// TIA Portal V17 export
// export: Created 2024-08-29T18:23:44.0966443Z, ExportSetting WithDefaults, DisplayName Totally Integrated Automation Portal, DisplayVersion V17 Update 7, DisplayName TIA Portal Openness, DisplayVersion V17 Update 7, DisplayName TIA Portal Version Control Interface, DisplayVersion V17, DisplayName SINAMICS Startdrive Advanced, DisplayVersion V17 SP2, DisplayName SINAMICS Startdrive G110M, G120, G120C, G120D, G120P, G115D, DisplayVersion V17 SP2, DisplayName SINAMICS Startdrive G130, G150, S120, S150, SINAMICS MV, S210, DisplayVersion V17 SP2, DisplayName STEP 7 Professional, DisplayVersion V17 Update 7, DisplayName STEP 7 Safety, DisplayVersion V17 Update 6, DisplayName WinCC Advanced / Unified PC, DisplayVersion V17 Update 7
FUNCTION "cylinderControl" : Void   // FC9, LAD
{ S7_Optimized_Access := 'TRUE' }
VERSION : 0.1
// stored: AutoNumber true, IsIECCheckEnabled false, SetENOAutomatically false, UDAEnableTagReadback false
   VAR_TEMP
      leftTrackReady : Bool;
      rightTrackReady : Bool;
      plasticBridgeReady : Bool;
      retractLocatingPinReady : Bool;
      enableCylinders : Bool;
      retractClampsReady : Bool;
   END_VAR
   VAR_TEMP   // added for the SCL form of the ladder/FBD networks
      _w1 : Bool;
   END_VAR
BEGIN

REGION Network 1: ENABLE CYLINDER GLOBAL
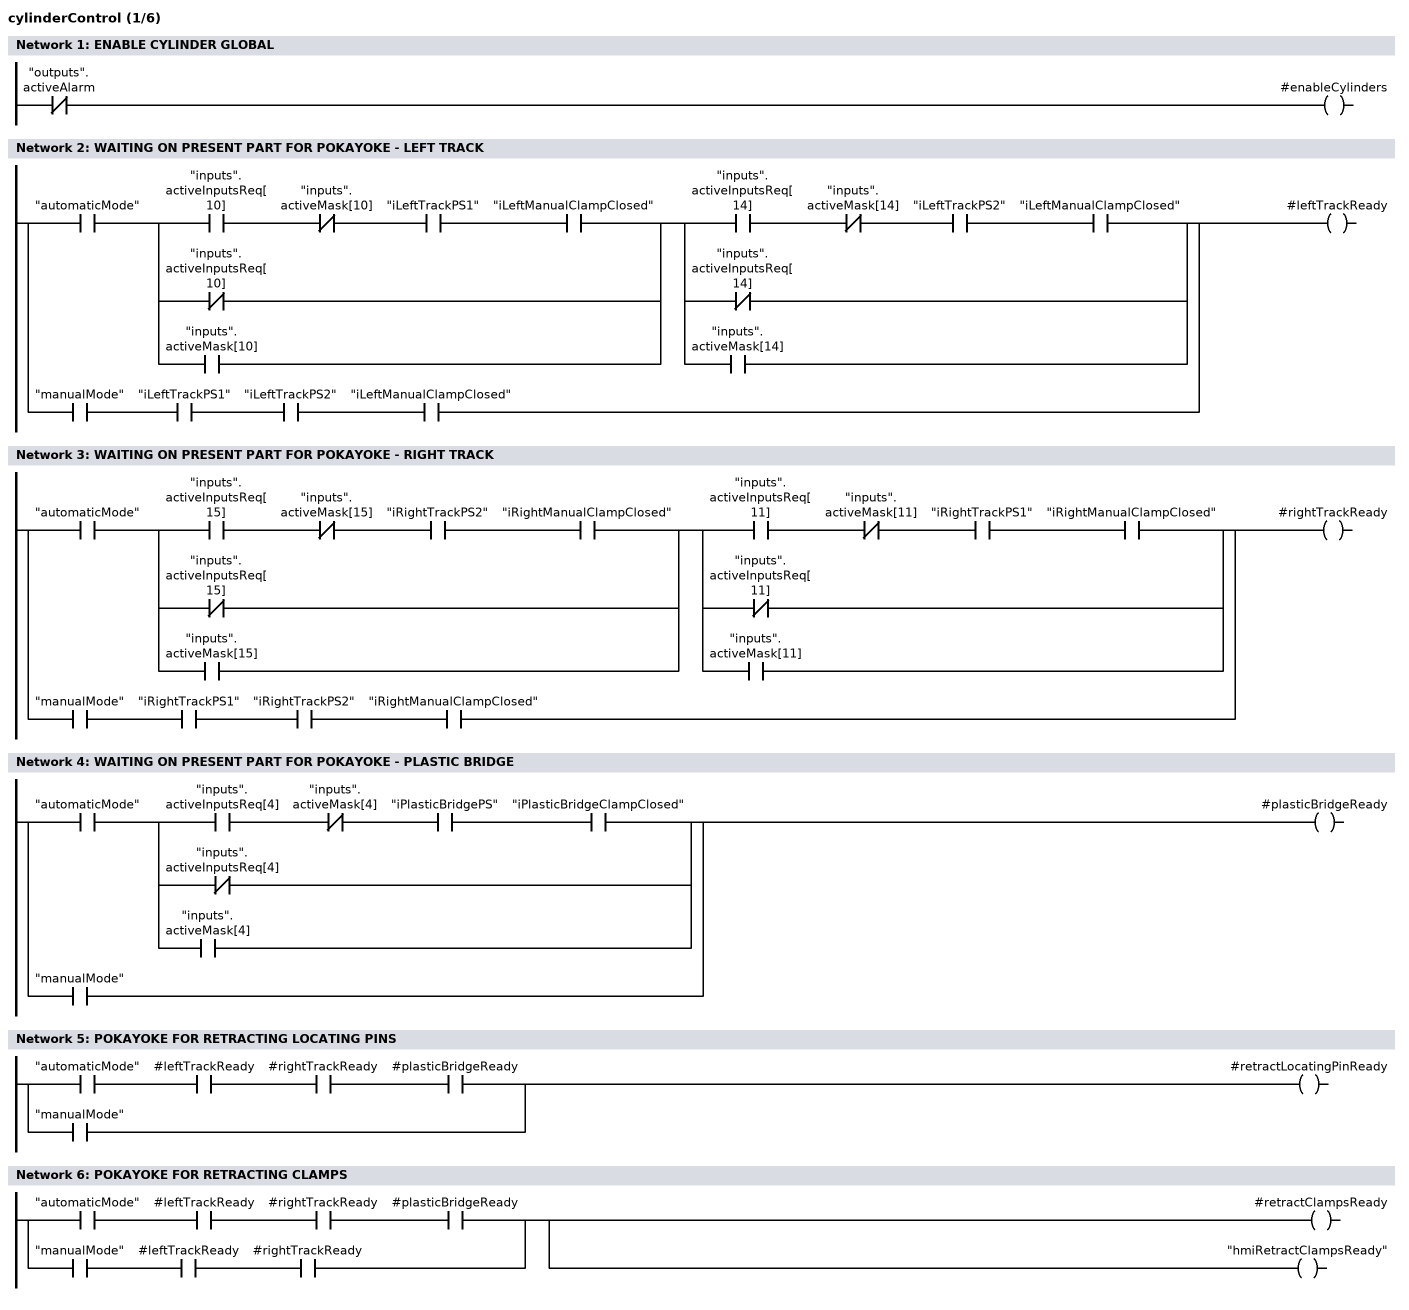
   RUNG wire#powerrail
      I_Contact( "outputs".activeAlarm )
      Coil( #enableCylinders )
   END_RUNG
   // the same network as SCL:
   #enableCylinders := NOT "outputs".activeAlarm;
END_REGION

REGION Network 2: WAITING ON PRESENT PART FOR POKAYOKE - LEFT TRACK
   RUNG wire#powerrail
      Contact( "automaticMode" )
      wire#w1
      Contact( "inputs".activeInputsReq[10] )
      I_Contact( "inputs".activeMask[10] )
      Contact( "iLeftTrackPS1" )
      Contact( "iLeftManualClampClosed" )
      wire#w2
      Contact( "inputs".activeInputsReq[14] )
      I_Contact( "inputs".activeMask[14] )
      Contact( "iLeftTrackPS2" )
      Contact( "iLeftManualClampClosed" )
      wire#w3
      Coil( #leftTrackReady )
   END_RUNG
   RUNG wire#w1
      I_Contact( "inputs".activeInputsReq[10] )
   END_RUNG wire#w2
   RUNG wire#w1
      Contact( "inputs".activeMask[10] )
   END_RUNG wire#w2
   RUNG wire#w2
      I_Contact( "inputs".activeInputsReq[14] )
   END_RUNG wire#w3
   RUNG wire#w2
      Contact( "inputs".activeMask[14] )
   END_RUNG wire#w3
   RUNG wire#powerrail
      Contact( "manualMode" )
      Contact( "iLeftTrackPS1" )
      Contact( "iLeftTrackPS2" )
      Contact( "iLeftManualClampClosed" )
   END_RUNG wire#w3
   // the same network as SCL:
   #leftTrackReady := ("automaticMode" AND (("inputs".activeInputsReq[10] AND NOT "inputs".activeMask[10] AND "iLeftTrackPS1" AND "iLeftManualClampClosed") OR NOT "inputs".activeInputsReq[10] OR "inputs".activeMask[10]) AND (("inputs".activeInputsReq[14] AND NOT "inputs".activeMask[14] AND "iLeftTrackPS2" AND "iLeftManualClampClosed") OR NOT "inputs".activeInputsReq[14] OR "inputs".activeMask[14])) OR ("manualMode" AND "iLeftTrackPS1" AND "iLeftTrackPS2" AND "iLeftManualClampClosed");
END_REGION

REGION Network 3: WAITING ON PRESENT PART FOR POKAYOKE - RIGHT TRACK
   RUNG wire#powerrail
      Contact( "automaticMode" )
      wire#w1
      Contact( "inputs".activeInputsReq[15] )
      I_Contact( "inputs".activeMask[15] )
      Contact( "iRightTrackPS2" )
      Contact( "iRightManualClampClosed" )
      wire#w2
      Contact( "inputs".activeInputsReq[11] )
      I_Contact( "inputs".activeMask[11] )
      Contact( "iRightTrackPS1" )
      Contact( "iRightManualClampClosed" )
      wire#w3
      Coil( #rightTrackReady )
   END_RUNG
   RUNG wire#w1
      I_Contact( "inputs".activeInputsReq[15] )
   END_RUNG wire#w2
   RUNG wire#w1
      Contact( "inputs".activeMask[15] )
   END_RUNG wire#w2
   RUNG wire#w2
      I_Contact( "inputs".activeInputsReq[11] )
   END_RUNG wire#w3
   RUNG wire#w2
      Contact( "inputs".activeMask[11] )
   END_RUNG wire#w3
   RUNG wire#powerrail
      Contact( "manualMode" )
      Contact( "iRightTrackPS1" )
      Contact( "iRightTrackPS2" )
      Contact( "iRightManualClampClosed" )
   END_RUNG wire#w3
   // the same network as SCL:
   #rightTrackReady := ("automaticMode" AND (("inputs".activeInputsReq[15] AND NOT "inputs".activeMask[15] AND "iRightTrackPS2" AND "iRightManualClampClosed") OR NOT "inputs".activeInputsReq[15] OR "inputs".activeMask[15]) AND (("inputs".activeInputsReq[11] AND NOT "inputs".activeMask[11] AND "iRightTrackPS1" AND "iRightManualClampClosed") OR NOT "inputs".activeInputsReq[11] OR "inputs".activeMask[11])) OR ("manualMode" AND "iRightTrackPS1" AND "iRightTrackPS2" AND "iRightManualClampClosed");
END_REGION

REGION Network 4: WAITING ON PRESENT PART FOR POKAYOKE - PLASTIC BRIDGE
   RUNG wire#powerrail
      Contact( "automaticMode" )
      wire#w1
      Contact( "inputs".activeInputsReq[4] )
      I_Contact( "inputs".activeMask[4] )
      Contact( "iPlasticBridgePS" )
      Contact( "iPlasticBridgeClampClosed" )
      wire#w2
      Coil( #plasticBridgeReady )
   END_RUNG
   RUNG wire#w1
      I_Contact( "inputs".activeInputsReq[4] )
   END_RUNG wire#w2
   RUNG wire#w1
      Contact( "inputs".activeMask[4] )
   END_RUNG wire#w2
   RUNG wire#powerrail
      Contact( "manualMode" )
   END_RUNG wire#w2
   // the same network as SCL:
   #plasticBridgeReady := ("automaticMode" AND (("inputs".activeInputsReq[4] AND NOT "inputs".activeMask[4] AND "iPlasticBridgePS" AND "iPlasticBridgeClampClosed") OR NOT "inputs".activeInputsReq[4] OR "inputs".activeMask[4])) OR "manualMode";
END_REGION

REGION Network 5: POKAYOKE FOR RETRACTING LOCATING PINS
   RUNG wire#powerrail
      Contact( "automaticMode" )
      Contact( #leftTrackReady )
      Contact( #rightTrackReady )
      Contact( #plasticBridgeReady )
      wire#w1
      Coil( #retractLocatingPinReady )
   END_RUNG
   RUNG wire#powerrail
      Contact( "manualMode" )
   END_RUNG wire#w1
   // the same network as SCL:
   #retractLocatingPinReady := ("automaticMode" AND #leftTrackReady AND #rightTrackReady AND #plasticBridgeReady) OR "manualMode";
END_REGION

REGION Network 6: POKAYOKE FOR RETRACTING CLAMPS
   RUNG wire#powerrail
      Contact( "automaticMode" )
      Contact( #leftTrackReady )
      Contact( #rightTrackReady )
      Contact( #plasticBridgeReady )
      wire#w1
      Coil( #retractClampsReady )
   END_RUNG
   RUNG wire#powerrail
      Contact( "manualMode" )
      Contact( #leftTrackReady )
      Contact( #rightTrackReady )
   END_RUNG wire#w1
   RUNG wire#w1
      Coil( "hmiRetractClampsReady" )
   END_RUNG
   // the same network as SCL:
   #retractClampsReady := ("automaticMode" AND #leftTrackReady AND #rightTrackReady AND #plasticBridgeReady) OR ("manualMode" AND #leftTrackReady AND #rightTrackReady);
   "hmiRetractClampsReady" := #retractClampsReady;
END_REGION

REGION Network 7: EXT CYL 1.- LEFT NEST LOCATING PIN EXTENDED
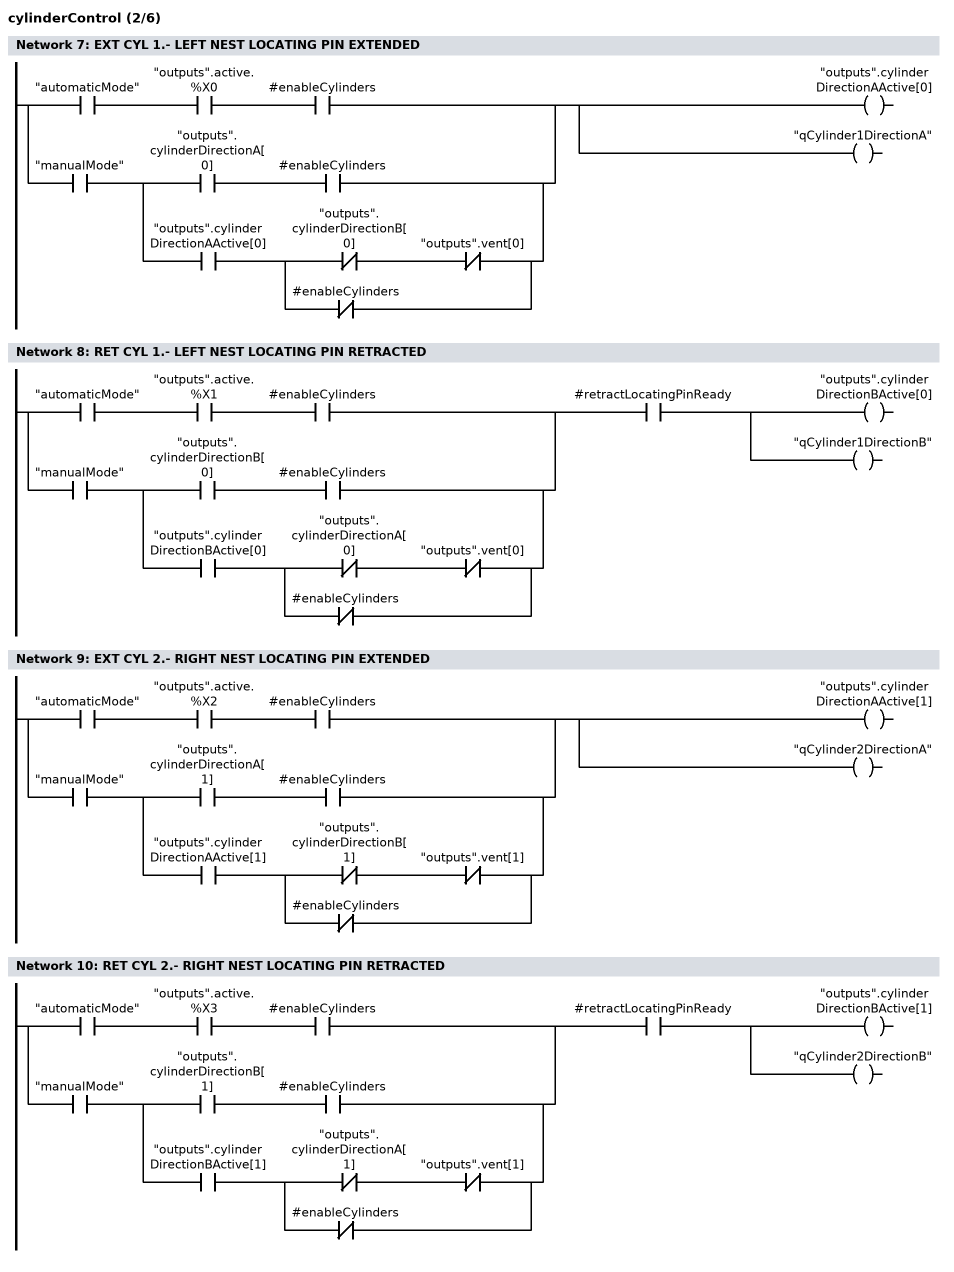
   RUNG wire#powerrail
      Contact( "automaticMode" )
      Contact( "outputs".active.%X0 )
      Contact( #enableCylinders )
      wire#w1
      Coil( "outputs".cylinderDirectionAActive[0] )
   END_RUNG
   RUNG wire#powerrail
      Contact( "manualMode" )
      wire#w2
      Contact( "outputs".cylinderDirectionA[0] )
      Contact( #enableCylinders )
   END_RUNG wire#w1
   RUNG wire#w2
      Contact( "outputs".cylinderDirectionAActive[0] )
      wire#w3
      I_Contact( "outputs".cylinderDirectionB[0] )
      I_Contact( "outputs".vent[0] )
   END_RUNG wire#w1
   RUNG wire#w3
      I_Contact( #enableCylinders )
   END_RUNG wire#w1
   RUNG wire#w1
      Coil( "qCylinder1DirectionA" )
   END_RUNG
   // the same network as SCL:
   #_w1 := ("automaticMode" AND "outputs".active.%X0 AND #enableCylinders) OR ("manualMode" AND (("outputs".cylinderDirectionA[0] AND #enableCylinders) OR ("outputs".cylinderDirectionAActive[0] AND ((NOT "outputs".cylinderDirectionB[0] AND NOT "outputs".vent[0]) OR NOT #enableCylinders))));
   "outputs".cylinderDirectionAActive[0] := ("automaticMode" AND "outputs".active.%X0 AND #enableCylinders) OR ("manualMode" AND (("outputs".cylinderDirectionA[0] AND #enableCylinders) OR ("outputs".cylinderDirectionAActive[0] AND ((NOT "outputs".cylinderDirectionB[0] AND NOT "outputs".vent[0]) OR NOT #enableCylinders))));
   "qCylinder1DirectionA" := #_w1;
END_REGION

REGION Network 8: RET CYL 1.- LEFT NEST LOCATING PIN RETRACTED
   RUNG wire#powerrail
      Contact( "automaticMode" )
      Contact( "outputs".active.%X1 )
      Contact( #enableCylinders )
      wire#w1
      Contact( #retractLocatingPinReady )
      wire#w4
      Coil( "outputs".cylinderDirectionBActive[0] )
   END_RUNG
   RUNG wire#powerrail
      Contact( "manualMode" )
      wire#w2
      Contact( "outputs".cylinderDirectionB[0] )
      Contact( #enableCylinders )
   END_RUNG wire#w1
   RUNG wire#w2
      Contact( "outputs".cylinderDirectionBActive[0] )
      wire#w3
      I_Contact( "outputs".cylinderDirectionA[0] )
      I_Contact( "outputs".vent[0] )
   END_RUNG wire#w1
   RUNG wire#w3
      I_Contact( #enableCylinders )
   END_RUNG wire#w1
   RUNG wire#w4
      Coil( "qCylinder1DirectionB" )
   END_RUNG
   // the same network as SCL:
   #_w1 := (("automaticMode" AND "outputs".active.%X1 AND #enableCylinders) OR ("manualMode" AND (("outputs".cylinderDirectionB[0] AND #enableCylinders) OR ("outputs".cylinderDirectionBActive[0] AND ((NOT "outputs".cylinderDirectionA[0] AND NOT "outputs".vent[0]) OR NOT #enableCylinders))))) AND #retractLocatingPinReady;
   "outputs".cylinderDirectionBActive[0] := (("automaticMode" AND "outputs".active.%X1 AND #enableCylinders) OR ("manualMode" AND (("outputs".cylinderDirectionB[0] AND #enableCylinders) OR ("outputs".cylinderDirectionBActive[0] AND ((NOT "outputs".cylinderDirectionA[0] AND NOT "outputs".vent[0]) OR NOT #enableCylinders))))) AND #retractLocatingPinReady;
   "qCylinder1DirectionB" := #_w1;
END_REGION

REGION Network 9: EXT CYL 2.- RIGHT NEST LOCATING PIN EXTENDED
   RUNG wire#powerrail
      Contact( "automaticMode" )
      Contact( "outputs".active.%X2 )
      Contact( #enableCylinders )
      wire#w1
      Coil( "outputs".cylinderDirectionAActive[1] )
   END_RUNG
   RUNG wire#powerrail
      Contact( "manualMode" )
      wire#w2
      Contact( "outputs".cylinderDirectionA[1] )
      Contact( #enableCylinders )
   END_RUNG wire#w1
   RUNG wire#w2
      Contact( "outputs".cylinderDirectionAActive[1] )
      wire#w3
      I_Contact( "outputs".cylinderDirectionB[1] )
      I_Contact( "outputs".vent[1] )
   END_RUNG wire#w1
   RUNG wire#w3
      I_Contact( #enableCylinders )
   END_RUNG wire#w1
   RUNG wire#w1
      Coil( "qCylinder2DirectionA" )
   END_RUNG
   // the same network as SCL:
   #_w1 := ("automaticMode" AND "outputs".active.%X2 AND #enableCylinders) OR ("manualMode" AND (("outputs".cylinderDirectionA[1] AND #enableCylinders) OR ("outputs".cylinderDirectionAActive[1] AND ((NOT "outputs".cylinderDirectionB[1] AND NOT "outputs".vent[1]) OR NOT #enableCylinders))));
   "outputs".cylinderDirectionAActive[1] := ("automaticMode" AND "outputs".active.%X2 AND #enableCylinders) OR ("manualMode" AND (("outputs".cylinderDirectionA[1] AND #enableCylinders) OR ("outputs".cylinderDirectionAActive[1] AND ((NOT "outputs".cylinderDirectionB[1] AND NOT "outputs".vent[1]) OR NOT #enableCylinders))));
   "qCylinder2DirectionA" := #_w1;
END_REGION

REGION Network 10: RET CYL 2.- RIGHT NEST LOCATING PIN RETRACTED
   RUNG wire#powerrail
      Contact( "automaticMode" )
      Contact( "outputs".active.%X3 )
      Contact( #enableCylinders )
      wire#w1
      Contact( #retractLocatingPinReady )
      wire#w4
      Coil( "outputs".cylinderDirectionBActive[1] )
   END_RUNG
   RUNG wire#powerrail
      Contact( "manualMode" )
      wire#w2
      Contact( "outputs".cylinderDirectionB[1] )
      Contact( #enableCylinders )
   END_RUNG wire#w1
   RUNG wire#w2
      Contact( "outputs".cylinderDirectionBActive[1] )
      wire#w3
      I_Contact( "outputs".cylinderDirectionA[1] )
      I_Contact( "outputs".vent[1] )
   END_RUNG wire#w1
   RUNG wire#w3
      I_Contact( #enableCylinders )
   END_RUNG wire#w1
   RUNG wire#w4
      Coil( "qCylinder2DirectionB" )
   END_RUNG
   // the same network as SCL:
   #_w1 := (("automaticMode" AND "outputs".active.%X3 AND #enableCylinders) OR ("manualMode" AND (("outputs".cylinderDirectionB[1] AND #enableCylinders) OR ("outputs".cylinderDirectionBActive[1] AND ((NOT "outputs".cylinderDirectionA[1] AND NOT "outputs".vent[1]) OR NOT #enableCylinders))))) AND #retractLocatingPinReady;
   "outputs".cylinderDirectionBActive[1] := (("automaticMode" AND "outputs".active.%X3 AND #enableCylinders) OR ("manualMode" AND (("outputs".cylinderDirectionB[1] AND #enableCylinders) OR ("outputs".cylinderDirectionBActive[1] AND ((NOT "outputs".cylinderDirectionA[1] AND NOT "outputs".vent[1]) OR NOT #enableCylinders))))) AND #retractLocatingPinReady;
   "qCylinder2DirectionB" := #_w1;
END_REGION

REGION Network 11: EXT CYL 3.- RIGHT TRACK CLAMP EXTENDED
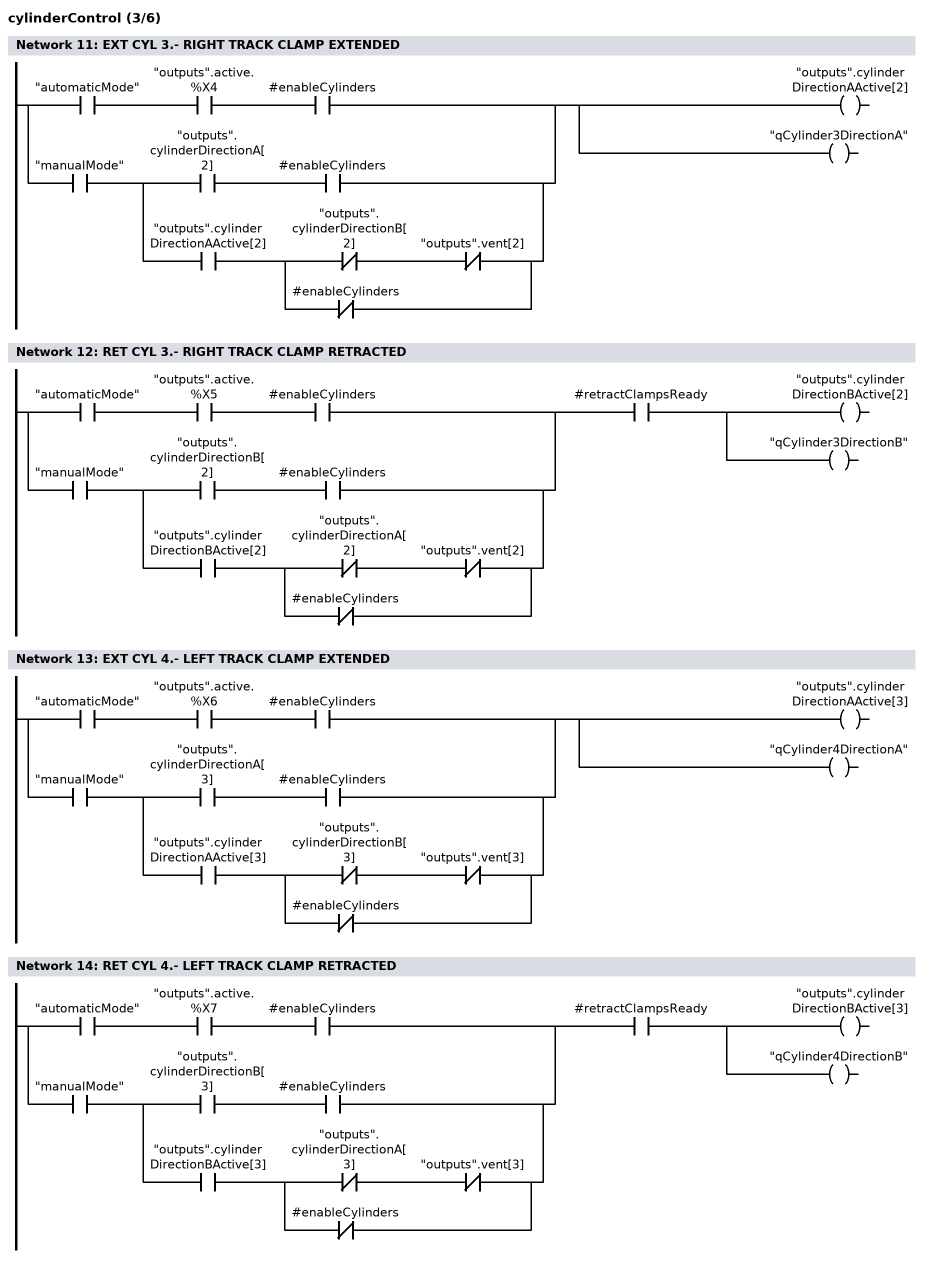
   RUNG wire#powerrail
      Contact( "automaticMode" )
      Contact( "outputs".active.%X4 )
      Contact( #enableCylinders )
      wire#w1
      Coil( "outputs".cylinderDirectionAActive[2] )
   END_RUNG
   RUNG wire#powerrail
      Contact( "manualMode" )
      wire#w2
      Contact( "outputs".cylinderDirectionA[2] )
      Contact( #enableCylinders )
   END_RUNG wire#w1
   RUNG wire#w2
      Contact( "outputs".cylinderDirectionAActive[2] )
      wire#w3
      I_Contact( "outputs".cylinderDirectionB[2] )
      I_Contact( "outputs".vent[2] )
   END_RUNG wire#w1
   RUNG wire#w3
      I_Contact( #enableCylinders )
   END_RUNG wire#w1
   RUNG wire#w1
      Coil( "qCylinder3DirectionA" )
   END_RUNG
   // the same network as SCL:
   #_w1 := ("automaticMode" AND "outputs".active.%X4 AND #enableCylinders) OR ("manualMode" AND (("outputs".cylinderDirectionA[2] AND #enableCylinders) OR ("outputs".cylinderDirectionAActive[2] AND ((NOT "outputs".cylinderDirectionB[2] AND NOT "outputs".vent[2]) OR NOT #enableCylinders))));
   "outputs".cylinderDirectionAActive[2] := ("automaticMode" AND "outputs".active.%X4 AND #enableCylinders) OR ("manualMode" AND (("outputs".cylinderDirectionA[2] AND #enableCylinders) OR ("outputs".cylinderDirectionAActive[2] AND ((NOT "outputs".cylinderDirectionB[2] AND NOT "outputs".vent[2]) OR NOT #enableCylinders))));
   "qCylinder3DirectionA" := #_w1;
END_REGION

REGION Network 12: RET CYL 3.- RIGHT TRACK CLAMP RETRACTED
   RUNG wire#powerrail
      Contact( "automaticMode" )
      Contact( "outputs".active.%X5 )
      Contact( #enableCylinders )
      wire#w1
      Contact( #retractClampsReady )
      wire#w4
      Coil( "outputs".cylinderDirectionBActive[2] )
   END_RUNG
   RUNG wire#powerrail
      Contact( "manualMode" )
      wire#w2
      Contact( "outputs".cylinderDirectionB[2] )
      Contact( #enableCylinders )
   END_RUNG wire#w1
   RUNG wire#w2
      Contact( "outputs".cylinderDirectionBActive[2] )
      wire#w3
      I_Contact( "outputs".cylinderDirectionA[2] )
      I_Contact( "outputs".vent[2] )
   END_RUNG wire#w1
   RUNG wire#w3
      I_Contact( #enableCylinders )
   END_RUNG wire#w1
   RUNG wire#w4
      Coil( "qCylinder3DirectionB" )
   END_RUNG
   // the same network as SCL:
   #_w1 := (("automaticMode" AND "outputs".active.%X5 AND #enableCylinders) OR ("manualMode" AND (("outputs".cylinderDirectionB[2] AND #enableCylinders) OR ("outputs".cylinderDirectionBActive[2] AND ((NOT "outputs".cylinderDirectionA[2] AND NOT "outputs".vent[2]) OR NOT #enableCylinders))))) AND #retractClampsReady;
   "outputs".cylinderDirectionBActive[2] := (("automaticMode" AND "outputs".active.%X5 AND #enableCylinders) OR ("manualMode" AND (("outputs".cylinderDirectionB[2] AND #enableCylinders) OR ("outputs".cylinderDirectionBActive[2] AND ((NOT "outputs".cylinderDirectionA[2] AND NOT "outputs".vent[2]) OR NOT #enableCylinders))))) AND #retractClampsReady;
   "qCylinder3DirectionB" := #_w1;
END_REGION

REGION Network 13: EXT CYL 4.- LEFT TRACK CLAMP EXTENDED
   RUNG wire#powerrail
      Contact( "automaticMode" )
      Contact( "outputs".active.%X6 )
      Contact( #enableCylinders )
      wire#w1
      Coil( "outputs".cylinderDirectionAActive[3] )
   END_RUNG
   RUNG wire#powerrail
      Contact( "manualMode" )
      wire#w2
      Contact( "outputs".cylinderDirectionA[3] )
      Contact( #enableCylinders )
   END_RUNG wire#w1
   RUNG wire#w2
      Contact( "outputs".cylinderDirectionAActive[3] )
      wire#w3
      I_Contact( "outputs".cylinderDirectionB[3] )
      I_Contact( "outputs".vent[3] )
   END_RUNG wire#w1
   RUNG wire#w3
      I_Contact( #enableCylinders )
   END_RUNG wire#w1
   RUNG wire#w1
      Coil( "qCylinder4DirectionA" )
   END_RUNG
   // the same network as SCL:
   #_w1 := ("automaticMode" AND "outputs".active.%X6 AND #enableCylinders) OR ("manualMode" AND (("outputs".cylinderDirectionA[3] AND #enableCylinders) OR ("outputs".cylinderDirectionAActive[3] AND ((NOT "outputs".cylinderDirectionB[3] AND NOT "outputs".vent[3]) OR NOT #enableCylinders))));
   "outputs".cylinderDirectionAActive[3] := ("automaticMode" AND "outputs".active.%X6 AND #enableCylinders) OR ("manualMode" AND (("outputs".cylinderDirectionA[3] AND #enableCylinders) OR ("outputs".cylinderDirectionAActive[3] AND ((NOT "outputs".cylinderDirectionB[3] AND NOT "outputs".vent[3]) OR NOT #enableCylinders))));
   "qCylinder4DirectionA" := #_w1;
END_REGION

REGION Network 14: RET CYL 4.- LEFT TRACK CLAMP RETRACTED
   RUNG wire#powerrail
      Contact( "automaticMode" )
      Contact( "outputs".active.%X7 )
      Contact( #enableCylinders )
      wire#w1
      Contact( #retractClampsReady )
      wire#w4
      Coil( "outputs".cylinderDirectionBActive[3] )
   END_RUNG
   RUNG wire#powerrail
      Contact( "manualMode" )
      wire#w2
      Contact( "outputs".cylinderDirectionB[3] )
      Contact( #enableCylinders )
   END_RUNG wire#w1
   RUNG wire#w2
      Contact( "outputs".cylinderDirectionBActive[3] )
      wire#w3
      I_Contact( "outputs".cylinderDirectionA[3] )
      I_Contact( "outputs".vent[3] )
   END_RUNG wire#w1
   RUNG wire#w3
      I_Contact( #enableCylinders )
   END_RUNG wire#w1
   RUNG wire#w4
      Coil( "qCylinder4DirectionB" )
   END_RUNG
   // the same network as SCL:
   #_w1 := (("automaticMode" AND "outputs".active.%X7 AND #enableCylinders) OR ("manualMode" AND (("outputs".cylinderDirectionB[3] AND #enableCylinders) OR ("outputs".cylinderDirectionBActive[3] AND ((NOT "outputs".cylinderDirectionA[3] AND NOT "outputs".vent[3]) OR NOT #enableCylinders))))) AND #retractClampsReady;
   "outputs".cylinderDirectionBActive[3] := (("automaticMode" AND "outputs".active.%X7 AND #enableCylinders) OR ("manualMode" AND (("outputs".cylinderDirectionB[3] AND #enableCylinders) OR ("outputs".cylinderDirectionBActive[3] AND ((NOT "outputs".cylinderDirectionA[3] AND NOT "outputs".vent[3]) OR NOT #enableCylinders))))) AND #retractClampsReady;
   "qCylinder4DirectionB" := #_w1;
END_REGION

REGION Network 15: EXT CYL 5.- SPARE
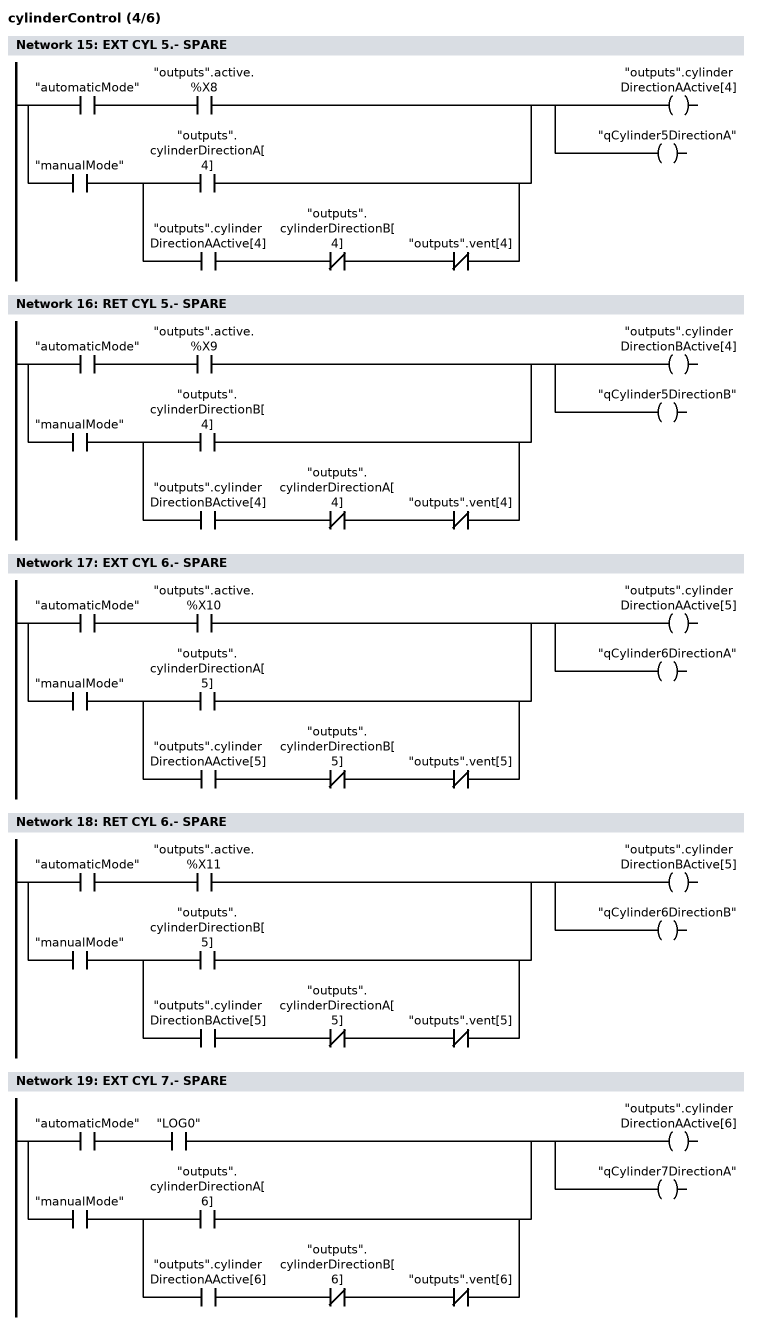
   RUNG wire#powerrail
      Contact( "automaticMode" )
      Contact( "outputs".active.%X8 )
      wire#w1
      Coil( "outputs".cylinderDirectionAActive[4] )
   END_RUNG
   RUNG wire#powerrail
      Contact( "manualMode" )
      wire#w2
      Contact( "outputs".cylinderDirectionA[4] )
   END_RUNG wire#w1
   RUNG wire#w2
      Contact( "outputs".cylinderDirectionAActive[4] )
      I_Contact( "outputs".cylinderDirectionB[4] )
      I_Contact( "outputs".vent[4] )
   END_RUNG wire#w1
   RUNG wire#w1
      Coil( "qCylinder5DirectionA" )
   END_RUNG
   // the same network as SCL:
   #_w1 := ("automaticMode" AND "outputs".active.%X8) OR ("manualMode" AND ("outputs".cylinderDirectionA[4] OR ("outputs".cylinderDirectionAActive[4] AND NOT "outputs".cylinderDirectionB[4] AND NOT "outputs".vent[4])));
   "outputs".cylinderDirectionAActive[4] := ("automaticMode" AND "outputs".active.%X8) OR ("manualMode" AND ("outputs".cylinderDirectionA[4] OR ("outputs".cylinderDirectionAActive[4] AND NOT "outputs".cylinderDirectionB[4] AND NOT "outputs".vent[4])));
   "qCylinder5DirectionA" := #_w1;
END_REGION

REGION Network 16: RET CYL 5.- SPARE
   RUNG wire#powerrail
      Contact( "automaticMode" )
      Contact( "outputs".active.%X9 )
      wire#w1
      Coil( "outputs".cylinderDirectionBActive[4] )
   END_RUNG
   RUNG wire#powerrail
      Contact( "manualMode" )
      wire#w2
      Contact( "outputs".cylinderDirectionB[4] )
   END_RUNG wire#w1
   RUNG wire#w2
      Contact( "outputs".cylinderDirectionBActive[4] )
      I_Contact( "outputs".cylinderDirectionA[4] )
      I_Contact( "outputs".vent[4] )
   END_RUNG wire#w1
   RUNG wire#w1
      Coil( "qCylinder5DirectionB" )
   END_RUNG
   // the same network as SCL:
   #_w1 := ("automaticMode" AND "outputs".active.%X9) OR ("manualMode" AND ("outputs".cylinderDirectionB[4] OR ("outputs".cylinderDirectionBActive[4] AND NOT "outputs".cylinderDirectionA[4] AND NOT "outputs".vent[4])));
   "outputs".cylinderDirectionBActive[4] := ("automaticMode" AND "outputs".active.%X9) OR ("manualMode" AND ("outputs".cylinderDirectionB[4] OR ("outputs".cylinderDirectionBActive[4] AND NOT "outputs".cylinderDirectionA[4] AND NOT "outputs".vent[4])));
   "qCylinder5DirectionB" := #_w1;
END_REGION

REGION Network 17: EXT CYL 6.- SPARE
   RUNG wire#powerrail
      Contact( "automaticMode" )
      Contact( "outputs".active.%X10 )
      wire#w1
      Coil( "outputs".cylinderDirectionAActive[5] )
   END_RUNG
   RUNG wire#powerrail
      Contact( "manualMode" )
      wire#w2
      Contact( "outputs".cylinderDirectionA[5] )
   END_RUNG wire#w1
   RUNG wire#w2
      Contact( "outputs".cylinderDirectionAActive[5] )
      I_Contact( "outputs".cylinderDirectionB[5] )
      I_Contact( "outputs".vent[5] )
   END_RUNG wire#w1
   RUNG wire#w1
      Coil( "qCylinder6DirectionA" )
   END_RUNG
   // the same network as SCL:
   #_w1 := ("automaticMode" AND "outputs".active.%X10) OR ("manualMode" AND ("outputs".cylinderDirectionA[5] OR ("outputs".cylinderDirectionAActive[5] AND NOT "outputs".cylinderDirectionB[5] AND NOT "outputs".vent[5])));
   "outputs".cylinderDirectionAActive[5] := ("automaticMode" AND "outputs".active.%X10) OR ("manualMode" AND ("outputs".cylinderDirectionA[5] OR ("outputs".cylinderDirectionAActive[5] AND NOT "outputs".cylinderDirectionB[5] AND NOT "outputs".vent[5])));
   "qCylinder6DirectionA" := #_w1;
END_REGION

REGION Network 18: RET CYL 6.- SPARE
   RUNG wire#powerrail
      Contact( "automaticMode" )
      Contact( "outputs".active.%X11 )
      wire#w1
      Coil( "outputs".cylinderDirectionBActive[5] )
   END_RUNG
   RUNG wire#powerrail
      Contact( "manualMode" )
      wire#w2
      Contact( "outputs".cylinderDirectionB[5] )
   END_RUNG wire#w1
   RUNG wire#w2
      Contact( "outputs".cylinderDirectionBActive[5] )
      I_Contact( "outputs".cylinderDirectionA[5] )
      I_Contact( "outputs".vent[5] )
   END_RUNG wire#w1
   RUNG wire#w1
      Coil( "qCylinder6DirectionB" )
   END_RUNG
   // the same network as SCL:
   #_w1 := ("automaticMode" AND "outputs".active.%X11) OR ("manualMode" AND ("outputs".cylinderDirectionB[5] OR ("outputs".cylinderDirectionBActive[5] AND NOT "outputs".cylinderDirectionA[5] AND NOT "outputs".vent[5])));
   "outputs".cylinderDirectionBActive[5] := ("automaticMode" AND "outputs".active.%X11) OR ("manualMode" AND ("outputs".cylinderDirectionB[5] OR ("outputs".cylinderDirectionBActive[5] AND NOT "outputs".cylinderDirectionA[5] AND NOT "outputs".vent[5])));
   "qCylinder6DirectionB" := #_w1;
END_REGION

REGION Network 19: EXT CYL 7.- SPARE
   RUNG wire#powerrail
      Contact( "automaticMode" )
      Contact( "LOG0" )
      wire#w1
      Coil( "outputs".cylinderDirectionAActive[6] )
   END_RUNG
   RUNG wire#powerrail
      Contact( "manualMode" )
      wire#w2
      Contact( "outputs".cylinderDirectionA[6] )
   END_RUNG wire#w1
   RUNG wire#w2
      Contact( "outputs".cylinderDirectionAActive[6] )
      I_Contact( "outputs".cylinderDirectionB[6] )
      I_Contact( "outputs".vent[6] )
   END_RUNG wire#w1
   RUNG wire#w1
      Coil( "qCylinder7DirectionA" )
   END_RUNG
   // the same network as SCL:
   #_w1 := ("automaticMode" AND "LOG0") OR ("manualMode" AND ("outputs".cylinderDirectionA[6] OR ("outputs".cylinderDirectionAActive[6] AND NOT "outputs".cylinderDirectionB[6] AND NOT "outputs".vent[6])));
   "outputs".cylinderDirectionAActive[6] := ("automaticMode" AND "LOG0") OR ("manualMode" AND ("outputs".cylinderDirectionA[6] OR ("outputs".cylinderDirectionAActive[6] AND NOT "outputs".cylinderDirectionB[6] AND NOT "outputs".vent[6])));
   "qCylinder7DirectionA" := #_w1;
END_REGION

REGION Network 20: RET CYL 7.- SPARE
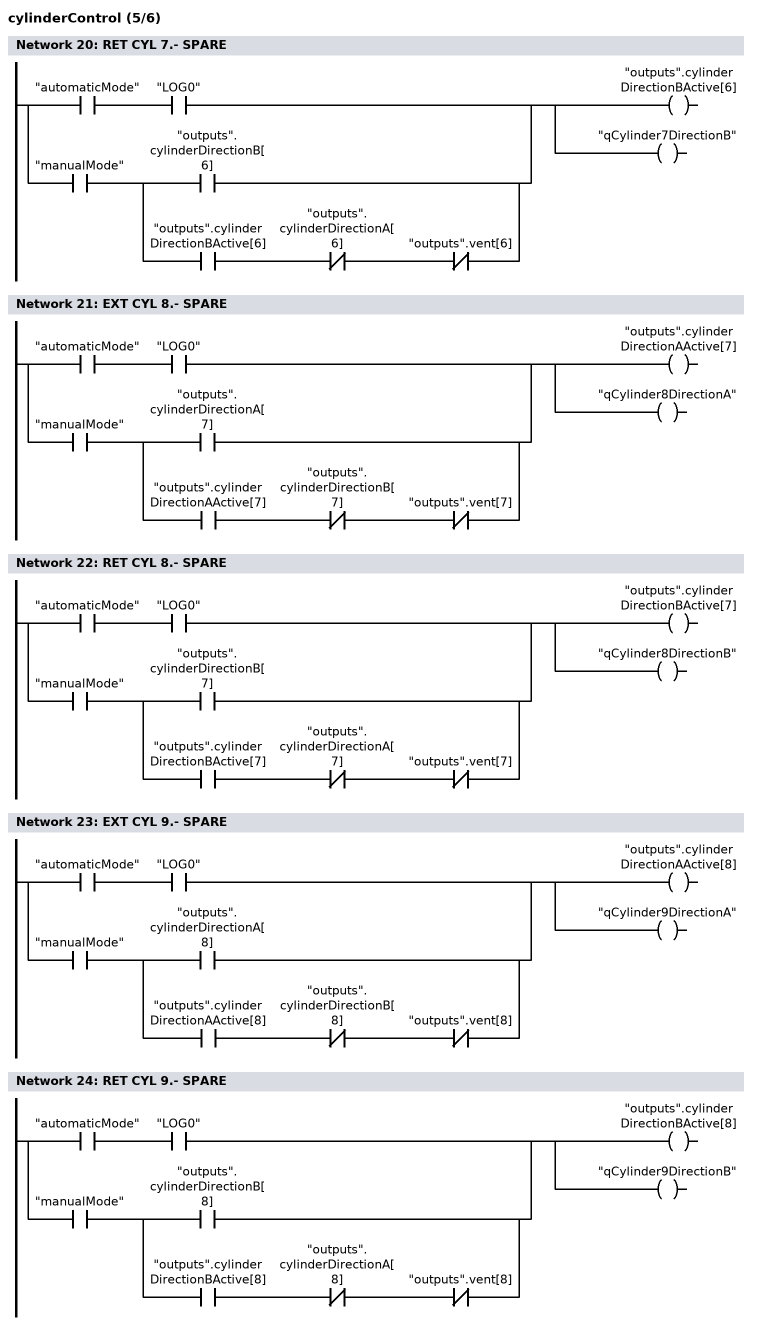
   RUNG wire#powerrail
      Contact( "automaticMode" )
      Contact( "LOG0" )
      wire#w1
      Coil( "outputs".cylinderDirectionBActive[6] )
   END_RUNG
   RUNG wire#powerrail
      Contact( "manualMode" )
      wire#w2
      Contact( "outputs".cylinderDirectionB[6] )
   END_RUNG wire#w1
   RUNG wire#w2
      Contact( "outputs".cylinderDirectionBActive[6] )
      I_Contact( "outputs".cylinderDirectionA[6] )
      I_Contact( "outputs".vent[6] )
   END_RUNG wire#w1
   RUNG wire#w1
      Coil( "qCylinder7DirectionB" )
   END_RUNG
   // the same network as SCL:
   #_w1 := ("automaticMode" AND "LOG0") OR ("manualMode" AND ("outputs".cylinderDirectionB[6] OR ("outputs".cylinderDirectionBActive[6] AND NOT "outputs".cylinderDirectionA[6] AND NOT "outputs".vent[6])));
   "outputs".cylinderDirectionBActive[6] := ("automaticMode" AND "LOG0") OR ("manualMode" AND ("outputs".cylinderDirectionB[6] OR ("outputs".cylinderDirectionBActive[6] AND NOT "outputs".cylinderDirectionA[6] AND NOT "outputs".vent[6])));
   "qCylinder7DirectionB" := #_w1;
END_REGION

REGION Network 21: EXT CYL 8.- SPARE
   RUNG wire#powerrail
      Contact( "automaticMode" )
      Contact( "LOG0" )
      wire#w1
      Coil( "outputs".cylinderDirectionAActive[7] )
   END_RUNG
   RUNG wire#powerrail
      Contact( "manualMode" )
      wire#w2
      Contact( "outputs".cylinderDirectionA[7] )
   END_RUNG wire#w1
   RUNG wire#w2
      Contact( "outputs".cylinderDirectionAActive[7] )
      I_Contact( "outputs".cylinderDirectionB[7] )
      I_Contact( "outputs".vent[7] )
   END_RUNG wire#w1
   RUNG wire#w1
      Coil( "qCylinder8DirectionA" )
   END_RUNG
   // the same network as SCL:
   #_w1 := ("automaticMode" AND "LOG0") OR ("manualMode" AND ("outputs".cylinderDirectionA[7] OR ("outputs".cylinderDirectionAActive[7] AND NOT "outputs".cylinderDirectionB[7] AND NOT "outputs".vent[7])));
   "outputs".cylinderDirectionAActive[7] := ("automaticMode" AND "LOG0") OR ("manualMode" AND ("outputs".cylinderDirectionA[7] OR ("outputs".cylinderDirectionAActive[7] AND NOT "outputs".cylinderDirectionB[7] AND NOT "outputs".vent[7])));
   "qCylinder8DirectionA" := #_w1;
END_REGION

REGION Network 22: RET CYL 8.- SPARE
   RUNG wire#powerrail
      Contact( "automaticMode" )
      Contact( "LOG0" )
      wire#w1
      Coil( "outputs".cylinderDirectionBActive[7] )
   END_RUNG
   RUNG wire#powerrail
      Contact( "manualMode" )
      wire#w2
      Contact( "outputs".cylinderDirectionB[7] )
   END_RUNG wire#w1
   RUNG wire#w2
      Contact( "outputs".cylinderDirectionBActive[7] )
      I_Contact( "outputs".cylinderDirectionA[7] )
      I_Contact( "outputs".vent[7] )
   END_RUNG wire#w1
   RUNG wire#w1
      Coil( "qCylinder8DirectionB" )
   END_RUNG
   // the same network as SCL:
   #_w1 := ("automaticMode" AND "LOG0") OR ("manualMode" AND ("outputs".cylinderDirectionB[7] OR ("outputs".cylinderDirectionBActive[7] AND NOT "outputs".cylinderDirectionA[7] AND NOT "outputs".vent[7])));
   "outputs".cylinderDirectionBActive[7] := ("automaticMode" AND "LOG0") OR ("manualMode" AND ("outputs".cylinderDirectionB[7] OR ("outputs".cylinderDirectionBActive[7] AND NOT "outputs".cylinderDirectionA[7] AND NOT "outputs".vent[7])));
   "qCylinder8DirectionB" := #_w1;
END_REGION

REGION Network 23: EXT CYL 9.- SPARE
   RUNG wire#powerrail
      Contact( "automaticMode" )
      Contact( "LOG0" )
      wire#w1
      Coil( "outputs".cylinderDirectionAActive[8] )
   END_RUNG
   RUNG wire#powerrail
      Contact( "manualMode" )
      wire#w2
      Contact( "outputs".cylinderDirectionA[8] )
   END_RUNG wire#w1
   RUNG wire#w2
      Contact( "outputs".cylinderDirectionAActive[8] )
      I_Contact( "outputs".cylinderDirectionB[8] )
      I_Contact( "outputs".vent[8] )
   END_RUNG wire#w1
   RUNG wire#w1
      Coil( "qCylinder9DirectionA" )
   END_RUNG
   // the same network as SCL:
   #_w1 := ("automaticMode" AND "LOG0") OR ("manualMode" AND ("outputs".cylinderDirectionA[8] OR ("outputs".cylinderDirectionAActive[8] AND NOT "outputs".cylinderDirectionB[8] AND NOT "outputs".vent[8])));
   "outputs".cylinderDirectionAActive[8] := ("automaticMode" AND "LOG0") OR ("manualMode" AND ("outputs".cylinderDirectionA[8] OR ("outputs".cylinderDirectionAActive[8] AND NOT "outputs".cylinderDirectionB[8] AND NOT "outputs".vent[8])));
   "qCylinder9DirectionA" := #_w1;
END_REGION

REGION Network 24: RET CYL 9.- SPARE
   RUNG wire#powerrail
      Contact( "automaticMode" )
      Contact( "LOG0" )
      wire#w1
      Coil( "outputs".cylinderDirectionBActive[8] )
   END_RUNG
   RUNG wire#powerrail
      Contact( "manualMode" )
      wire#w2
      Contact( "outputs".cylinderDirectionB[8] )
   END_RUNG wire#w1
   RUNG wire#w2
      Contact( "outputs".cylinderDirectionBActive[8] )
      I_Contact( "outputs".cylinderDirectionA[8] )
      I_Contact( "outputs".vent[8] )
   END_RUNG wire#w1
   RUNG wire#w1
      Coil( "qCylinder9DirectionB" )
   END_RUNG
   // the same network as SCL:
   #_w1 := ("automaticMode" AND "LOG0") OR ("manualMode" AND ("outputs".cylinderDirectionB[8] OR ("outputs".cylinderDirectionBActive[8] AND NOT "outputs".cylinderDirectionA[8] AND NOT "outputs".vent[8])));
   "outputs".cylinderDirectionBActive[8] := ("automaticMode" AND "LOG0") OR ("manualMode" AND ("outputs".cylinderDirectionB[8] OR ("outputs".cylinderDirectionBActive[8] AND NOT "outputs".cylinderDirectionA[8] AND NOT "outputs".vent[8])));
   "qCylinder9DirectionB" := #_w1;
END_REGION

REGION Network 25: EXT CYL 10.- SPARE **
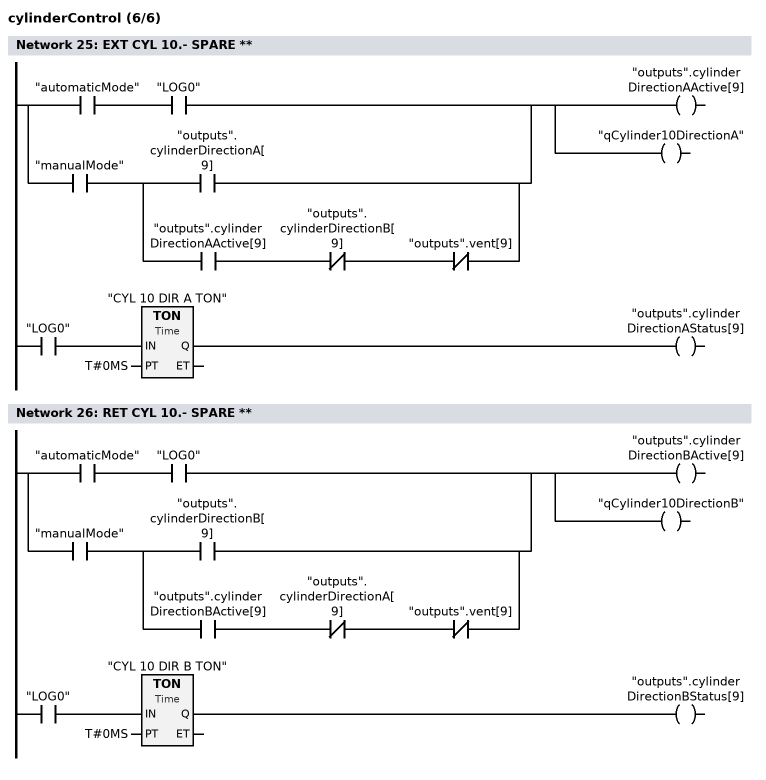
   RUNG wire#powerrail
      Contact( "automaticMode" )
      Contact( "LOG0" )
      wire#w1
      Coil( "outputs".cylinderDirectionAActive[9] )
   END_RUNG
   RUNG wire#powerrail
      Contact( "manualMode" )
      wire#w2
      Contact( "outputs".cylinderDirectionA[9] )
   END_RUNG wire#w1
   RUNG wire#w2
      Contact( "outputs".cylinderDirectionAActive[9] )
      I_Contact( "outputs".cylinderDirectionB[9] )
      I_Contact( "outputs".vent[9] )
   END_RUNG wire#w1
   RUNG wire#w1
      Coil( "qCylinder10DirectionA" )
   END_RUNG
   RUNG wire#powerrail
      Contact( "LOG0" )
      { S7_Templates := "time_type := Time" } "CYL 10 DIR A TON".TON(pt := T#0MS, et =>)
      Coil( "outputs".cylinderDirectionAStatus[9] )
   END_RUNG
   // the same network as SCL:
   #_w1 := ("automaticMode" AND "LOG0") OR ("manualMode" AND ("outputs".cylinderDirectionA[9] OR ("outputs".cylinderDirectionAActive[9] AND NOT "outputs".cylinderDirectionB[9] AND NOT "outputs".vent[9])));
   "outputs".cylinderDirectionAActive[9] := ("automaticMode" AND "LOG0") OR ("manualMode" AND ("outputs".cylinderDirectionA[9] OR ("outputs".cylinderDirectionAActive[9] AND NOT "outputs".cylinderDirectionB[9] AND NOT "outputs".vent[9])));
   "qCylinder10DirectionA" := #_w1;
   "CYL 10 DIR A TON".TON(IN := "LOG0", PT := T#0MS);
   "outputs".cylinderDirectionAStatus[9] := "CYL 10 DIR A TON".Q;
END_REGION

REGION Network 26: RET CYL 10.- SPARE **
   RUNG wire#powerrail
      Contact( "automaticMode" )
      Contact( "LOG0" )
      wire#w1
      Coil( "outputs".cylinderDirectionBActive[9] )
   END_RUNG
   RUNG wire#powerrail
      Contact( "manualMode" )
      wire#w2
      Contact( "outputs".cylinderDirectionB[9] )
   END_RUNG wire#w1
   RUNG wire#w2
      Contact( "outputs".cylinderDirectionBActive[9] )
      I_Contact( "outputs".cylinderDirectionA[9] )
      I_Contact( "outputs".vent[9] )
   END_RUNG wire#w1
   RUNG wire#w1
      Coil( "qCylinder10DirectionB" )
   END_RUNG
   RUNG wire#powerrail
      Contact( "LOG0" )
      { S7_Templates := "time_type := Time" } "CYL 10 DIR B TON".TON(pt := T#0MS, et =>)
      Coil( "outputs".cylinderDirectionBStatus[9] )
   END_RUNG
   // the same network as SCL:
   #_w1 := ("automaticMode" AND "LOG0") OR ("manualMode" AND ("outputs".cylinderDirectionB[9] OR ("outputs".cylinderDirectionBActive[9] AND NOT "outputs".cylinderDirectionA[9] AND NOT "outputs".vent[9])));
   "outputs".cylinderDirectionBActive[9] := ("automaticMode" AND "LOG0") OR ("manualMode" AND ("outputs".cylinderDirectionB[9] OR ("outputs".cylinderDirectionBActive[9] AND NOT "outputs".cylinderDirectionA[9] AND NOT "outputs".vent[9])));
   "qCylinder10DirectionB" := #_w1;
   "CYL 10 DIR B TON".TON(IN := "LOG0", PT := T#0MS);
   "outputs".cylinderDirectionBStatus[9] := "CYL 10 DIR B TON".Q;
END_REGION
END_FUNCTION
